// TIA Portal V19 export
ORGANIZATION_BLOCK "Startup"   // OB100, FBD, Startup
TITLE = "Complete Restart"
{ S7_Optimized_Access := 'TRUE' }
// stored: SetENOAutomatically false
   VAR_INPUT
      LostRetentive : Bool;   // True if retentive data are lost
      LostRTC : Bool;   // True if date and time are lost
   END_VAR
BEGIN

REGION Network 1: Set point for automatic mode LC1 och CV1
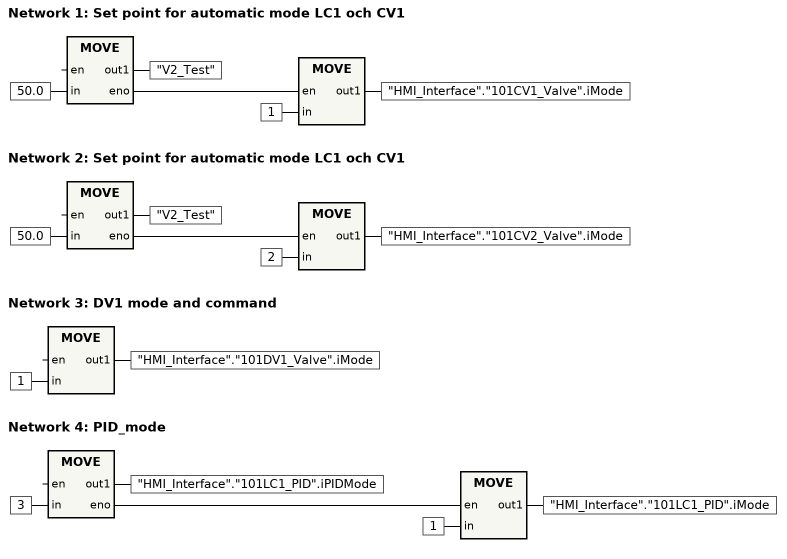
   "V2_Test" := 50.0;
   "HMI_Interface"."101CV1_Valve".iMode := 1;
END_REGION

REGION Network 2: Set point for automatic mode LC1 och CV1
   "V2_Test" := 50.0;
   "HMI_Interface"."101CV2_Valve".iMode := 2;
END_REGION

REGION Network 3: DV1 mode and command
   "HMI_Interface"."101DV1_Valve".iMode := 1;
END_REGION

REGION Network 4: PID_mode
   "HMI_Interface"."101LC1_PID".iPIDMode := 3;
   "HMI_Interface"."101LC1_PID".iMode := 1;
END_REGION
END_ORGANIZATION_BLOCK
